{attribute 'GeneratedUsingTerminal: EK1100-0000-0018'}
{attribute addProperty BoxType "EK1100-0000-0018"}
{attribute addProperty Id "Beckhoff_ELM3xxxEK1122Beckhoff_ELM3xxxEK1122_1A0BF0352A_0001_ELM3002_0000_0016ELM3002_B416BFEF50A_0002_ELM3002_0000_0017ELM3002_B416BFEF50A_0003_ELM3002_0000_0018ELM3002_B416BFEF50A_0004_ELM3004_0000_0016ELM3004_9E251EA472A_0005_ELM3004_0000_0017ELM3004_9E251EA472A_0006_ELM3004_0000_0018ELM3004_9E251EA472A_0007_ELM3004_0000_0019ELM3004_9E251EA472"}
{attribute addProperty CRC "832849192"}
{attribute addProperty Size "440"}
TYPE Beckhoff_ELM3xxx_31A44528 EXTENDS EK1100_1FC0878B :
STRUCT
	{attribute addProperty Name "Beckhoff_ELM3xxxEK1122"}
	Beckhoff_ELM3xxxEK1122 : Beckhoff_ELM3xxxEK1122_1A0BF035;
	{attribute addProperty Name "A_0001_ELM3002_0000_0016"}
	A_0001_ELM3002_0000_0016 : ELM3002_B416BFEF;
	{attribute addProperty Name "A_0002_ELM3002_0000_0017"}
	A_0002_ELM3002_0000_0017 : ELM3002_B416BFEF;
	{attribute addProperty Name "A_0003_ELM3002_0000_0018"}
	A_0003_ELM3002_0000_0018 : ELM3002_B416BFEF;
	{attribute addProperty Name "A_0004_ELM3004_0000_0016"}
	A_0004_ELM3004_0000_0016 : ELM3004_9E251EA4;
	{attribute addProperty Name "A_0005_ELM3004_0000_0017"}
	A_0005_ELM3004_0000_0017 : ELM3004_9E251EA4;
	{attribute addProperty Name "A_0006_ELM3004_0000_0018"}
	A_0006_ELM3004_0000_0018 : ELM3004_9E251EA4;
	{attribute addProperty Name "A_0007_ELM3004_0000_0019"}
	A_0007_ELM3004_0000_0019 : ELM3004_9E251EA4;
END_STRUCT
END_TYPE

(* stored: Version 1.2.0.0, ProductVersion 3.1.4024.9
   DUT Beckhoff_ELM3xxx_31A44528: Id {c873ef04-848a-47f5-ad51-d69e0a8c1f06} *)
